{attribute 'GeneratedUsingTerminal: AX8108-0100-0101-0101'}
{attribute addProperty BoxType "AX8108-0100-0101-0101"}
{attribute addProperty Id "Power_supply_controlwordAT %Q*UINT2"}
{attribute addProperty CRC "1695495302"}
{attribute addProperty Size "2"}
TYPE DeviceMain_Outputs_650F3486 EXTENDS OutputBase_10CEE7DE :
STRUCT
	{attribute addProperty Name "Power_supply_controlword"}
	Power_supply_controlword AT %Q* : UINT;
END_STRUCT
END_TYPE

(* stored: Version 1.2.0.0, ProductVersion 3.1.4024.9
   DUT DeviceMain_Outputs_650F3486: Id {5101cc5e-4d57-41f3-a80c-f1a490f8ad5c} *)
